TYPE ST_Inverter_UgridStatusWord :
STRUCT
	//Ugrid Status Word
		b_ChargeControlActive			: BOOL;
		b_InternalChargingSwitchStatus	: BOOL;
		b_MCBcontrol					: BOOL;
		b_MCBStatus						: BOOL;
		b_RunEnabled					: BOOL;
		b_DriveReady					: BOOL;
		b_AFEmodeActive					: BOOL;
		b_IslandModeActive				: BOOL;
		b_MicrogridModeActive			: BOOL;
		b_RunRequestActive				: BOOL;
		b_DriveInRunState				: BOOL;
		b_FaultActive					: BOOL;
		b_SynchronizedToD7				: BOOL;
		b_D7MeasurementsOK				: BOOL;	
END_STRUCT
END_TYPE

(* stored: Version 1.1.0.1, ProductVersion 3.1.4026.18
   DUT ST_Inverter_UgridStatusWord: Id {43e59534-e251-475f-841f-59cb818df532} *)
